FUNCTION_BLOCK AR_TO_AUDI (* Composite FB for converting AR (REAL) adapter to AUDI (UDINT) adapter — numeric conversion (value-preserving cast; narrowing may truncate, widening/sign-extension is safe). *)
  (* Standard: 61499-2; Description: Copyright (c) 2026 HR Agrartechnik GmbH This program and the accompanying materials are made available under the terms of the Eclipse Public License 2.0 which is available at https://www.eclipse.org/legal/epl-2.0/ SPDX-License-Identifier: EPL-2.0 *)
  (* Version 1.0, 2026-02-17, Franz Höpfinger, HR Agrartechnik GmbH *)
  PACKAGE adapter::conversion::unidirectional;
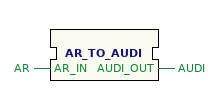
  SOCKETS
    AR_IN : adapter::types::unidirectional::AR; (* REAL Adapter Input *)
  END_SOCKETS
  PLUGS
    AUDI_OUT : adapter::types::unidirectional::AUDI; (* UDINT Adapter Output *)
  END_PLUGS
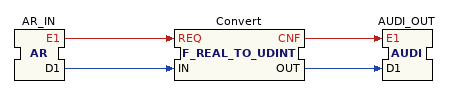
  FBS
    Convert : iec61131::conversion::F_REAL_TO_UDINT;
  END_FBS
  EVENT_CONNECTIONS
    AR_IN.E1 TO Convert.REQ;
    Convert.CNF TO AUDI_OUT.E1;
  END_CONNECTIONS
  DATA_CONNECTIONS
    AR_IN.D1 TO Convert.IN;
    Convert.OUT TO AUDI_OUT.D1;
  END_CONNECTIONS
END_FUNCTION_BLOCK
